// TIA Portal V17 export
// export: Created 2023-02-13T11:16:10.0685453Z, ExportSetting WithDefaults, DisplayName Totally Integrated Automation Portal, DisplayVersion V17, DisplayName TIA Portal Openness, DisplayVersion V17, DisplayName TIA Portal Teamcenter Gateway, DisplayVersion V17, DisplayName TIA Portal Version Control Interface, DisplayVersion V17, DisplayName SINAMICS Startdrive Advanced, DisplayVersion V17, DisplayName SINAMICS Startdrive G130, G150, S120, S150, SINAMICS MV, S210, DisplayVersion V17, DisplayName SINAMICS Startdrive G110M, G120, G120C, G120D, G120P, G115D, DisplayVersion V17, DisplayName STEP 7 Professional, DisplayVersion V17, DisplayName STEP 7 Safety, DisplayVersion V17, DisplayName WinCC Professional, DisplayVersion V17
DATA_BLOCK "AlarmFlowColletor"   // DB217
VERSION : 0.1
// stored: AutoNumber false, DBAccessibleFromOPCUA true, DBAccessibleFromWebserver true, InstanceOfName Alarm Flow Collector, InstanceOfType FB
"Alarm Flow Collector"
   // VAR_INPUT
   //    Reset : Bool;
   // END_VAR
   // VAR
   //    alwaysON : Bool;
   // END_VAR
   // VAR RETAIN
   //    Param : Struct
   //       min_Flow : Struct
   //          ChiliAwetan1 : Real;
   //          ChiliAwetan2 : Real;
   //          ChiliAwetan3 : Real;
   //          Tomato : Real;
   //          ChiliFresh1 : Real;
   //          ChiliFresh2 : Real;
   //          ChiliFresh3 : Real;
   //          Garlic : Real;
   //          HW : Real;
   //          Vinegar : Real;
   //          Sugar : Real;
   //          Salt : Real;
   //          ProWater : Real;
   //          Homomixer : Real;
   //       END_STRUCT;
   //       timerMon : Struct
   //          ChiliAwetan1 : TON_TIME;
   //          ChiliAwetan2 : TON_TIME;
   //          ChiliAwetan3 : TON_TIME;
   //          Tomato : TON_TIME;
   //          ChiliFresh1 : TON_TIME;
   //          ChiliFresh2 : TON_TIME;
   //          ChiliFresh3 : TON_TIME;
   //          Garlic : TON_TIME;
   //          HW : TON_TIME;
   //          Vinegar : TON_TIME;
   //          Sugar : TON_TIME;
   //          Salt : TON_TIME;
   //          ProWater : TON_TIME;
   //          Homomixer : TON_TIME;
   //       END_STRUCT;
   //    END_STRUCT;
   // END_VAR
   // VAR
   //    AlarmFlow_Blend : Word;
   // END_VAR
BEGIN
END_DATA_BLOCK
